// TIA Portal V15.1 export
// export: Created 2024-06-21T08:41:08.4201455Z, ExportSetting WithDefaults, DisplayName Totally Integrated Automation Portal, DisplayVersion V15.1 Update 5, DisplayName TIA Portal Openness, DisplayVersion V15.1 Update 5, DisplayName SINAMICS Startdrive Advanced, DisplayVersion V15.1, DisplayName G130, G150, S120, S150, SINAMICS MV, S210, DisplayVersion V15.1, DisplayName G110M, G120, G120C, G120D, G120P, DisplayVersion V15.1, DisplayName STEP 7 Professional, DisplayVersion V15.1 Update 5, DisplayName STEP 7 Safety, DisplayVersion V15.1, DisplayName WinCC Professional, DisplayVersion V15.1 Update 5, DisplayName SIMATIC Visualization Architect, DisplayVersion V15.1
FUNCTION "LGB10CharToDInt" : Int   // FC6600, SCL
{ S7_Optimized_Access := 'TRUE' }
VERSION : 0.1
// stored: AutoNumber false, IsIECCheckEnabled false, SetENOAutomatically False, UDAEnableTagReadback false
   VAR_INPUT
      I_char1 : Char;
      I_char2 : Char;
      I_char3 : Char;
      I_char4 : Char;
      I_char5 : Char;
      I_char6 : Char;
      I_char7 : Char;
      I_char8 : Char;
      I_char9 : Char;
      I_char10 : Char;
   END_VAR
   VAR_OUTPUT
      O_Dint : DInt;
      O_Error : Bool;
      O_ErrorNr : Int;
   END_VAR
   VAR_TEMP
      Str1 : String[1];
      Str2 : String[1];
      Str3 : String[1];
      Str4 : String[1];
      Str5 : String[1];
      Str6 : String[1];
      Str7 : String[1];
      Str8 : String[1];
      Str9 : String[1];
      Str10 : String[1];
      Str : String;
      conv_char1 : Char;
      conv_char2 : Char;
      conv_char3 : Char;
      conv_char4 : Char;
      conv_char5 : Char;
      conv_char6 : Char;
      conv_char7 : Char;
      conv_char8 : Char;
      conv_char9 : Char;
      conv_char10 : Char;
      t_char1 : Char;
      t_char2 : Char;
      t_char3 : Char;
      t_char4 : Char;
      t_char5 : Char;
      t_char6 : Char;
      t_char7 : Char;
      t_char8 : Char;
      t_char9 : Char;
      t_char10 : Char;
      t_Error : Int;
   END_VAR
BEGIN
   REGION INITIALISATION 

   #t_Error := 0;
   #O_Error := false;
   #O_ErrorNr := 0;

   END_REGION

   REGION Check if carachter is a number
       IF #I_char1 = '$00' THEN
           #conv_char1 := '0';
       ELSE
           #conv_char1 := #I_char1;
       END_IF;

       IF #I_char2 = '$00' THEN
           #conv_char2 := '0';
       ELSE
           #conv_char2 := #I_char2;
       END_IF;

       IF #I_char3 = '$00' THEN
           #conv_char3 := '0';
       ELSE
           #conv_char3 := #I_char3;
       END_IF;

       IF #I_char4 = '$00' THEN
           #conv_char4 := '0';
       ELSE
           #conv_char4 := #I_char4;
       END_IF;

       IF #I_char5 = '$00' THEN
           #conv_char5 := '0';
       ELSE
           #conv_char5 := #I_char5;
       END_IF;

       IF #I_char6 = '$00' THEN
           #conv_char6 := '0';
       ELSE
           #conv_char6 := #I_char6;
       END_IF;

       IF #I_char7 = '$00' THEN
           #conv_char7 := '0';
       ELSE
           #conv_char7 := #I_char7;
       END_IF;

       IF #I_char8 = '$00' THEN
           #conv_char8 := '0';
       ELSE
           #conv_char8 := #I_char8;
       END_IF;

       IF #I_char9 = '$00' THEN
           #conv_char9 := '0';
       ELSE
           #conv_char9 := #I_char9;
       END_IF;

       IF #I_char10 = '$00' THEN
           #conv_char10 := '0';
       ELSE
           #conv_char10 := #I_char10;
       END_IF;

       IF CHAR_TO_INT(#conv_char1) >= 48 AND CHAR_TO_INT(#conv_char1) <= 57 THEN
           #t_char1 := #conv_char1;
       ELSE
           #t_char1 := '0';
           #t_Error := 1;
       END_IF;
       IF CHAR_TO_INT(#conv_char2) >= 48 AND CHAR_TO_INT(#conv_char2) <= 57 THEN
           #t_char2 := #conv_char2;
       ELSE
           #t_char2 := '0';
           #t_Error := 2;
       END_IF;
       IF CHAR_TO_INT(#conv_char3) >= 48 AND CHAR_TO_INT(#conv_char3) <= 57 THEN
           #t_char3 := #conv_char3;
       ELSE
           #t_char3 := '0';
           #t_Error := 3;
       END_IF;
       IF CHAR_TO_INT(#conv_char4) >= 48 AND CHAR_TO_INT(#conv_char4) <= 57 THEN
           #t_char4 := #conv_char4;
       ELSE
           #t_char4 := '0';
           #t_Error := 4;
       END_IF;
       IF CHAR_TO_INT(#conv_char5) >= 48 AND CHAR_TO_INT(#conv_char5) <= 57 THEN
           #t_char5 := #conv_char5;
       ELSE
           #t_char5 := '0';
           #t_Error := 5;
       END_IF;
       IF CHAR_TO_INT(#conv_char6) >= 48 AND CHAR_TO_INT(#conv_char6) <= 57 THEN
           #t_char6 := #conv_char6;
       ELSE
           #t_char6 := '0';
           #t_Error := 6;
       END_IF;
       IF CHAR_TO_INT(#conv_char7) >= 48 AND CHAR_TO_INT(#conv_char7) <= 57 THEN
           #t_char7 := #conv_char7;
       ELSE
           #t_char7 := '0';
           #t_Error := 7;
       END_IF;
       IF CHAR_TO_INT(#conv_char8) >= 48 AND CHAR_TO_INT(#conv_char8) <= 57 THEN
           #t_char8 := #conv_char8;
       ELSE
           #t_char8 := '0';
           #t_Error := 8;
       END_IF;
       IF CHAR_TO_INT(#conv_char9) >= 48 AND CHAR_TO_INT(#conv_char9) <= 57 THEN
           #t_char9 := #conv_char9;
       ELSE
           #t_char9 := '0';
           #t_Error := 9;
       END_IF;
       IF CHAR_TO_INT(#conv_char10) >= 48 AND CHAR_TO_INT(#conv_char10) <= 57 THEN
           #t_char10 := #conv_char10;
       ELSE
           #t_char10 := '0';
           #t_Error := 10;
       END_IF;

   END_REGION

   REGION When no fault Change charachters TO String AND finaly TO a DInt
       IF #t_Error = 0 THEN

           #Str1 := CHAR_TO_STRING(#t_char1);
           #Str2 := CHAR_TO_STRING(#t_char2);
           #Str3 := CHAR_TO_STRING(#t_char3);
           #Str4 := CHAR_TO_STRING(#t_char4);
           #Str5 := CHAR_TO_STRING(#t_char5);
           #Str6 := CHAR_TO_STRING(#t_char6);
           #Str7 := CHAR_TO_STRING(#t_char7);
           #Str8 := CHAR_TO_STRING(#t_char8);
           #Str9 := CHAR_TO_STRING(#t_char9);
           #Str10 := CHAR_TO_STRING(#t_char10);

           #Str := CONCAT(IN1 := #Str1, IN2 := #Str2, IN3 := #Str3, IN4 := #Str4, IN5 := #Str5, IN6 := #Str6, IN7 := #Str7, IN8 := #Str8, IN9 := #Str9, IN10 := #Str10);
           #O_Dint := STRING_TO_DINT(#Str);

       ELSE //When fault write 0 and set errorbit high

           #O_Dint := 0;
           #O_ErrorNr := #t_Error;
           #O_Error := FALSE;

       END_IF;
   END_REGION

   #LGB10CharToDInt := 100;
END_FUNCTION
